(* IEC 61131-3 sources: plc-st-test/test/fixtures, 6 files *)

(* ---- types.st ---- *)
TYPE
  EColor : (Red, Green := 3, Blue);
  TPoint : STRUCT
    x : INT;
    y : INT := 5;
    color : EColor;
  END_STRUCT;
END_TYPE

(* ---- dup_a.st ---- *)
FUNCTION_BLOCK FB_Dup
  VAR
    a : INT;
  END_VAR
END_FUNCTION_BLOCK

(* ---- dup_b.st ---- *)
FUNCTION_BLOCK FB_Dup
  VAR
    b : BOOL;
  END_VAR
END_FUNCTION_BLOCK

(* ---- missing_endif.st ---- *)
FUNCTION_BLOCK FB_B
VAR
    x : INT;
END_VAR
    IF x > 0 THEN
        x := x + 1;
END_FUNCTION_BLOCK

(* ---- missing_semicolon.st ---- *)
FUNCTION_BLOCK FB_C
VAR
    x : INT;
END_VAR
    IF x > 0 THEN
        x := x + 1
    END_IF;
END_FUNCTION_BLOCK

(* ---- valid_fb.st ---- *)
FUNCTION_BLOCK FB_A
VAR
    x : INT;
END_VAR
    x := 1;
END_FUNCTION_BLOCK
